// Mitsubishi GX Works2 project: mcEx01   PLC: Q02/Q02H

PROGRAM MAIN
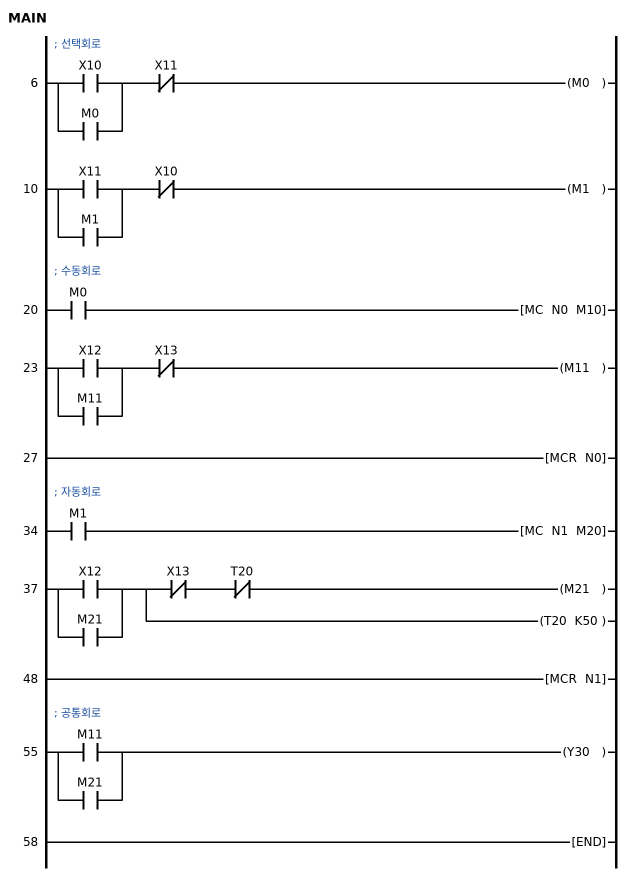
; 선택회로
6     LD      X10
      OR      M0
      ANI     X11
      OUT     M0
10    LD      X11
      OR      M1
      ANI     X10
      OUT     M1
; 수동회로
20    LD      M0
      MC      N0 M10
23    LD      X12
      OR      M11
      ANI     X13
      OUT     M11
27    MCR     N0
; 자동회로
34    LD      M1
      MC      N1 M20
37    LD      X12
      OR      M21
      MPS
      ANI     X13
      ANI     T20
      OUT     M21
      MPP
      OUT     T20 K50
48    MCR     N1
; 공통회로
55    LD      M11
      OR      M21
      OUT     Y30
58    END
END_PROGRAM
